# B&R Automation Studio project MotionTestBenchMaster (part 17)

### HMI_PAM_3.typ
```iecst
(*HMI_PAM_3 Database for Filler PLC*)
(*Author = ????*)
(*DB Version : 0.00*)
(*File Version : 3.23*)

TYPE
        HMI_PAM_3_Type:     STRUCT
                            _000 : REAL; (*SEAMER FERRUM - Seamer rinse: Hot water temperature [°C]*)
                            _001 : REAL; (*SEAMER FERRUM - Spare *)
                            _002 : REAL; (*SEAMER FERRUM - Spare *)
                            _003 : REAL; (*SEAMER FERRUM - Spare *)
                            _004 : REAL; (*SEAMER FERRUM - Spare *)
                            _005 : REAL; (*SEAMER FERRUM - Spare *)
                            _006 : REAL; (*SEAMER FERRUM - Spare *)
                            _007 : REAL; (*SEAMER FERRUM - Spare *)
                            _008 : REAL; (*SEAMER FERRUM - Spare *)
                            _009 : REAL; (*SEAMER FERRUM - Spare *)
                            _010 : REAL; (*SEAMER FERRUM - Machine Speed on seamer cleaning [c/h]*)
                            _011 : REAL; (*SEAMER FERRUM - Spare *)
                            _012 : REAL; (*SEAMER FERRUM - Spare *)
                            _013 : REAL; (*SEAMER FERRUM - Spare *)
                            _014 : REAL; (*SEAMER FERRUM - Spare *)
                            _015 : REAL; (*SEAMER FERRUM - Spare *)
                            _016 : REAL; (*SEAMER FERRUM - Spare *)
                            _017 : REAL; (*SEAMER FERRUM - Spare *)
                            _018 : REAL; (*SEAMER FERRUM - Spare *)
                            _019 : REAL; (*SEAMER FERRUM - Spare *)
                            _020 : REAL; (*SEAMER FERRUM - Spare *)
                            _021 : REAL; (*SEAMER FERRUM - Spare *)
                            _022 : REAL; (*SEAMER FERRUM - Spare *)
                            _023 : REAL; (*SEAMER FERRUM - Spare *)
                            _024 : REAL; (*SEAMER FERRUM - Spare *)
                            _025 : REAL; (*SEAMER FERRUM - Spare *)
                            _026 : REAL; (*SEAMER FERRUM - Spare *)
                            _027 : REAL; (*SEAMER FERRUM - Spare *)
                            _028 : REAL; (*SEAMER FERRUM - Spare *)
                            _029 : REAL; (*SEAMER FERRUM - Spare *)
                            _030 : REAL; (*SEAMER FERRUM - Spare *)
                            _031 : REAL; (*SEAMER FERRUM - Spare *)
                            _032 : REAL; (*SEAMER FERRUM - Spare *)
                            _033 : REAL; (*SEAMER FERRUM - Spare *)
                            _034 : REAL; (*SEAMER FERRUM - Spare *)
                            _035 : REAL; (*SEAMER FERRUM - Spare *)
                            _036 : REAL; (*SEAMER FERRUM - Spare *)
                            _037 : REAL; (*SEAMER FERRUM - Spare *)
                            _038 : REAL; (*SEAMER FERRUM - Spare *)
                            _039 : REAL; (*SEAMER FERRUM - Spare *)
                            _040 : REAL; (*SEAMER FERRUM - Spare *)
                            _041 : REAL; (*SEAMER FERRUM - Spare *)
                            _042 : REAL; (*SEAMER FERRUM - Spare *)
                            _043 : REAL; (*SEAMER FERRUM - Spare *)
                            _044 : REAL; (*SEAMER FERRUM - Spare *)
                            _045 : REAL; (*SEAMER FERRUM - Spare *)
                            _046 : REAL; (*SEAMER FERRUM - Spare *)
                            _047 : REAL; (*SEAMER FERRUM - Spare *)
                            _048 : REAL; (*SEAMER FERRUM - Spare *)
                            _049 : REAL; (*SEAMER FERRUM - Spare *)
                            _050 : REAL; (*SEAMER FERRUM - Spare *)
                            _051 : REAL; (*SEAMER FERRUM - Spare *)
                            _052 : REAL; (*SEAMER FERRUM - Spare *)
                            _053 : REAL; (*SEAMER FERRUM - Spare *)
                            _054 : REAL; (*SEAMER FERRUM - Spare *)
                            _055 : REAL; (*SEAMER FERRUM - Spare *)
                            _056 : REAL; (*SEAMER FERRUM - Spare *)
                            _057 : REAL; (*SEAMER FERRUM - Spare *)
                            _058 : REAL; (*SEAMER FERRUM - Spare *)
                            _059 : REAL; (*SEAMER FERRUM - Spare *)
                            _060 : REAL; (*SEAMER FERRUM - Spare *)
                            _061 : REAL; (*SEAMER FERRUM - Spare *)
                            _062 : REAL; (*SEAMER FERRUM - Spare *)
                            _063 : REAL; (*SEAMER FERRUM - Spare *)
                            _064 : REAL; (*SEAMER FERRUM - Spare *)
                            _065 : REAL; (*SEAMER FERRUM - Spare *)
                            _066 : REAL; (*SEAMER FERRUM - Spare *)
                            _067 : REAL; (*SEAMER FERRUM - Spare *)
                            _068 : REAL; (*SEAMER FERRUM - Spare *)
                            _069 : REAL; (*SEAMER FERRUM - Spare *)
                            _070 : REAL; (*SEAMER FERRUM - Spare *)
                            _071 : REAL; (*SEAMER FERRUM - Spare *)
                            _072 : REAL; (*SEAMER FERRUM - Spare *)
                            _073 : REAL; (*SEAMER FERRUM - Spare *)
                            _074 : REAL; (*SEAMER FERRUM - Spare *)
                            _075 : REAL; (*SEAMER FERRUM - Spare *)
                            _076 : REAL; (*SEAMER FERRUM - Spare *)
                            _077 : REAL; (*SEAMER FERRUM - Spare *)
                            _078 : REAL; (*SEAMER FERRUM - Spare *)
                            _079 : REAL; (*SEAMER FERRUM - Spare *)
                            _080 : REAL; (*SEAMER FERRUM - Spare *)
                            _081 : REAL; (*SEAMER FERRUM - Spare *)
                            _082 : REAL; (*SEAMER FERRUM - Spare *)
                            _083 : REAL; (*SEAMER FERRUM - Spare *)
                            _084 : REAL; (*SEAMER FERRUM - Spare *)
                            _085 : REAL; (*SEAMER FERRUM - Spare *)
                            _086 : REAL; (*SEAMER FERRUM - Spare *)
                            _087 : REAL; (*SEAMER FERRUM - Spare *)
                            _088 : REAL; (*SEAMER FERRUM - Spare *)
                            _089 : REAL; (*SEAMER FERRUM - Spare *)
                            _090 : REAL; (*SEAMER FERRUM - Spare *)
                            _091 : REAL; (*SEAMER FERRUM - Spare *)
                            _092 : REAL; (*SEAMER FERRUM - Spare *)
                            _093 : REAL; (*SEAMER FERRUM - Spare *)
                            _094 : REAL; (*SEAMER FERRUM - Spare *)
                            _095 : REAL; (*SEAMER FERRUM - Spare *)
                            _096 : REAL; (*SEAMER FERRUM - Spare *)
                            _097 : REAL; (*SEAMER FERRUM - Spare *)
                            _098 : REAL; (*SEAMER FERRUM - Spare *)
                            _099 : REAL; (*SEAMER FERRUM - Spare *)
                            _100 : REAL; (*SEAMER CFT - Seamer Lubrication *)
                            _101 : REAL; (*SEAMER CFT - Seamer Roll Lubrication *)
                            _102 : REAL; (*SEAMER CFT - Seamer Star Washing Time [s]*)
                            _103 : REAL; (*SEAMER CFT - Seamer Washing Time [s]*)
                            _104 : REAL; (*SEAMER CFT - Low Lubrication Cycle Aft Was *)
                            _105 : REAL; (*SEAMER CFT - Low Lubrication Cycle *)
                            _106 : REAL; (*SEAMER CFT - Lubrication Cycle Aft Was *)
                            _107 : REAL; (*SEAMER CFT - Rol Lubric Cycle *)
                            _108 : REAL; (*SEAMER CFT - N Timer *)
                            _109 : REAL; (*SEAMER CFT - Timer Value *)
                            _110 : REAL; (*SEAMER CFT - Spare *)
                            _111 : REAL; (*SEAMER CFT - Spare *)
                            _112 : REAL; (*SEAMER CFT - Roll_Lubrication_Enable *)
                            _113 : REAL; (*SEAMER CFT - Star Washing Enable *)
                            _114 : REAL; (*SEAMER CFT - Spare *)
                            _115 : REAL; (*SEAMER CFT - Spare *)
                            _116 : REAL; (*SEAMER CFT - Spare *)
                            _117 : REAL; (*SEAMER CFT - Spare *)
                            _118 : REAL; (*SEAMER CFT - Spare *)
                            _119 : REAL; (*SEAMER CFT - Spare *)
                            _120 : REAL; (*SEAMER CFT - Spare *)
                            _121 : REAL; (*SEAMER CFT - Spare *)
                            _122 : REAL; (*SEAMER CFT - Spare *)
                            _123 : REAL; (*SEAMER CFT - Spare *)
                            _124 : REAL; (*SEAMER CFT - Spare *)
                            _125 : REAL; (*SEAMER CFT - Spare *)
                            _126 : REAL; (*SEAMER CFT - Spare *)
                            _127 : REAL; (*SEAMER CFT - Spare *)
                            _128 : REAL; (*SEAMER CFT - Spare *)
                            _129 : REAL; (*SEAMER CFT - Spare *)
                            _130 : REAL; (*SEAMER CFT - Spare *)
                            _131 : REAL; (*SEAMER CFT - Spare *)
                            _132 : REAL; (*SEAMER CFT - Spare *)
                            _133 : REAL; (*SEAMER CFT - Spare *)
                            _134 : REAL; (*SEAMER CFT - Spare *)
                            _135 : REAL; (*SEAMER CFT - Spare *)
                            _136 : REAL; (*SEAMER CFT - Spare *)
                            _137 : REAL; (*SEAMER CFT - Spare *)
                            _138 : REAL; (*SEAMER CFT - Spare *)
                            _139 : REAL; (*SEAMER CFT - Spare *)
                            _140 : REAL; (*SEAMER CFT - Spare *)
                            _141 : REAL; (*SEAMER CFT - Spare *)
                            _142 : REAL; (*SEAMER CFT - Spare *)
                            _143 : REAL; (*SEAMER CFT - Spare *)
                            _144 : REAL; (*SEAMER CFT - Spare *)
                            _145 : REAL; (*SEAMER CFT - Spare *)
                            _146 : REAL; (*SEAMER CFT - Spare *)
                            _147 : REAL; (*SEAMER CFT - Spare *)
                            _148 : REAL; (*SEAMER CFT - Spare *)
                            _149 : REAL; (*SEAMER CFT - Spare *)
                            _150 : REAL; (*SEAMER CFT - Spare *)
                            _151 : REAL; (*SEAMER CFT - Spare *)
                            _152 : REAL; (*SEAMER CFT - Spare *)
                            _153 : REAL; (*SEAMER CFT - Spare *)
                            _154 : REAL; (*SEAMER CFT - Spare *)
                            _155 : REAL; (*SEAMER CFT - Spare *)
                            _156 : REAL; (*SEAMER CFT - Spare *)
                            _157 : REAL; (*SEAMER CFT - Spare *)
                            _158 : REAL; (*SEAMER CFT - Spare *)
                            _159 : REAL; (*SEAMER CFT - Spare *)
                            _160 : REAL; (*SEAMER CFT - Spare *)
                            _161 : REAL; (*SEAMER CFT - Spare *)
                            _162 : REAL; (*SEAMER CFT - Spare *)
                            _163 : REAL; (*SEAMER CFT - Spare *)
                            _164 : REAL; (*SEAMER CFT - Spare *)
                            _165 : REAL; (*SEAMER CFT - Spare *)
                            _166 : REAL; (*SEAMER CFT - Spare *)
                            _167 : REAL; (*SEAMER CFT - Spare *)
                            _168 : REAL; (*SEAMER CFT - Spare *)
                            _169 : REAL; (*SEAMER CFT - Spare *)
                            _170 : REAL; (*SEAMER CFT - Spare *)
                            _171 : REAL; (*SEAMER CFT - Spare *)
                            _172 : REAL; (*SEAMER CFT - Spare *)
                            _173 : REAL; (*SEAMER CFT - Spare *)
                            _174 : REAL; (*SEAMER CFT - Spare *)
                            _175 : REAL; (*SEAMER CFT - Spare *)
                            _176 : REAL; (*SEAMER CFT - Spare *)
                            _177 : REAL; (*SEAMER CFT - Spare *)
                            _178 : REAL; (*SEAMER CFT - Spare *)
                            _179 : REAL; (*SEAMER CFT - Spare *)
                            _180 : REAL; (*SEAMER CFT - Spare *)
                            _181 : REAL; (*SEAMER CFT - Spare *)
                            _182 : REAL; (*SEAMER CFT - Spare *)
                            _183 : REAL; (*SEAMER CFT - Spare *)
                            _184 : REAL; (*SEAMER CFT - Spare *)
                            _185 : REAL; (*SEAMER CFT - Spare *)
                            _186 : REAL; (*SEAMER CFT - Spare *)
                            _187 : REAL; (*SEAMER CFT - Spare *)
                            _188 : REAL; (*SEAMER CFT - Spare *)
                            _189 : REAL; (*SEAMER CFT - Spare *)
                            _190 : REAL; (*SEAMER CFT - Spare *)
                            _191 : REAL; (*SEAMER CFT - Spare *)
                            _192 : REAL; (*SEAMER CFT - Spare *)
                            _193 : REAL; (*SEAMER CFT - Spare *)
                            _194 : REAL; (*SEAMER CFT - Spare *)
                            _195 : REAL; (*SEAMER CFT - Spare *)
                            _196 : REAL; (*SEAMER CFT - Spare *)
                            _197 : REAL; (*SEAMER CFT - Spare *)
                            _198 : REAL; (*SEAMER CFT - Spare *)
                            _199 : REAL; (*SEAMER CFT - Spare *)
                            _200 : REAL; (*SEAMER ANGELUS - Seamer rinse: Hot water temperature [°C]*)
                            _201 : REAL; (*SEAMER ANGELUS - Spare *)
                            _202 : REAL; (*SEAMER ANGELUS - Spare *)
                            _203 : REAL; (*SEAMER ANGELUS - Spare *)
                            _204 : REAL; (*SEAMER ANGELUS - Spare *)
                            _205 : REAL; (*SEAMER ANGELUS - Spare *)
                            _206 : REAL; (*SEAMER ANGELUS - Spare *)
                            _207 : REAL; (*SEAMER ANGELUS - Spare *)
                            _208 : REAL; (*SEAMER ANGELUS - Spare *)
                            _209 : REAL; (*SEAMER ANGELUS - Spare *)
                            _210 : REAL; (*SEAMER ANGELUS - Machine Speed on seamer cleaning [c/h]*)
                            _211 : REAL; (*SEAMER ANGELUS - Spare *)
                            _212 : REAL; (*SEAMER ANGELUS - Spare *)
                            _213 : REAL; (*SEAMER ANGELUS - Spare *)
                            _214 : REAL; (*SEAMER ANGELUS - Spare *)
                            _215 : REAL; (*SEAMER ANGELUS - Spare *)
                            _216 : REAL; (*SEAMER ANGELUS - Spare *)
                            _217 : REAL; (*SEAMER ANGELUS - Spare *)
                            _218 : REAL; (*SEAMER ANGELUS - Spare *)
                            _219 : REAL; (*SEAMER ANGELUS - Spare *)
                            _220 : REAL; (*SEAMER ANGELUS - Spare *)
                            _221 : REAL; (*SEAMER ANGELUS - Spare *)
                            _222 : REAL; (*SEAMER ANGELUS - Spare *)
                            _223 : REAL; (*SEAMER ANGELUS - Spare *)
                            _224 : REAL; (*SEAMER ANGELUS - Spare *)
                            _225 : REAL; (*SEAMER ANGELUS - Spare *)
                            _226 : REAL; (*SEAMER ANGELUS - Spare *)
                            _227 : REAL; (*SEAMER ANGELUS - Spare *)
                            _228 : REAL; (*SEAMER ANGELUS - Spare *)
                            _229 : REAL; (*SEAMER ANGELUS - Spare *)
                            _230 : REAL; (*SEAMER ANGELUS - Spare *)
                            _231 : REAL; (*SEAMER ANGELUS - Spare *)
                            _232 : REAL; (*SEAMER ANGELUS - Spare *)
                            _233 : REAL; (*SEAMER ANGELUS - Spare *)
                            _234 : REAL; (*SEAMER ANGELUS - Spare *)
                            _235 : REAL; (*SEAMER ANGELUS - Spare *)
                            _236 : REAL; (*SEAMER ANGELUS - Spare *)
                            _237 : REAL; (*SEAMER ANGELUS - Spare *)
                            _238 : REAL; (*SEAMER ANGELUS - Spare *)
                            _239 : REAL; (*SEAMER ANGELUS - Spare *)
                            _240 : REAL; (*SEAMER ANGELUS - Spare *)
                            _241 : REAL; (*SEAMER ANGELUS - Spare *)
                            _242 : REAL; (*SEAMER ANGELUS - Spare *)
                            _243 : REAL; (*SEAMER ANGELUS - Spare *)
                            _244 : REAL; (*SEAMER ANGELUS - Spare *)
                            _245 : REAL; (*SEAMER ANGELUS - Spare *)
                            _246 : REAL; (*SEAMER ANGELUS - Spare *)
                            _247 : REAL; (*SEAMER ANGELUS - Spare *)
                            _248 : REAL; (*SEAMER ANGELUS - Spare *)
                            _249 : REAL; (*SEAMER ANGELUS - Spare *)
                            _250 : REAL; (*SEAMER ANGELUS - Spare *)
                            _251 : REAL; (*SEAMER ANGELUS - Spare *)
                            _252 : REAL; (*SEAMER ANGELUS - Spare *)
                            _253 : REAL; (*SEAMER ANGELUS - Spare *)
                            _254 : REAL; (*SEAMER ANGELUS - Spare *)
                            _255 : REAL; (*SEAMER ANGELUS - Spare *)
                            _256 : REAL; (*SEAMER ANGELUS - Spare *)
                            _257 : REAL; (*SEAMER ANGELUS - Spare *)
                            _258 : REAL; (*SEAMER ANGELUS - Spare *)
                            _259 : REAL; (*SEAMER ANGELUS - Spare *)
                            _260 : REAL; (*SEAMER ANGELUS - Spare *)
                            _261 : REAL; (*SEAMER ANGELUS - Spare *)
                            _262 : REAL; (*SEAMER ANGELUS - Spare *)
                            _263 : REAL; (*SEAMER ANGELUS - Spare *)
                            _264 : REAL; (*SEAMER ANGELUS - Spare *)
                            _265 : REAL; (*SEAMER ANGELUS - Spare *)
                            _266 : REAL; (*SEAMER ANGELUS - Spare *)
                            _267 : REAL; (*SEAMER ANGELUS - Spare *)
                            _268 : REAL; (*SEAMER ANGELUS - Spare *)
                            _269 : REAL; (*SEAMER ANGELUS - Spare *)
                            _270 : REAL; (*SEAMER ANGELUS - Spare *)
                            _271 : REAL; (*SEAMER ANGELUS - Spare *)
                            _272 : REAL; (*SEAMER ANGELUS - Spare *)
                            _273 : REAL; (*SEAMER ANGELUS - Spare *)
                            _274 : REAL; (*SEAMER ANGELUS - Spare *)
                            _275 : REAL; (*SEAMER ANGELUS - Spare *)
                            _276 : REAL; (*SEAMER ANGELUS - Spare *)
                            _277 : REAL; (*SEAMER ANGELUS - Spare *)
                            _278 : REAL; (*SEAMER ANGELUS - Spare *)
                            _279 : REAL; (*SEAMER ANGELUS - Spare *)
                            _280 : REAL; (*SEAMER ANGELUS - Spare *)
                            _281 : REAL; (*SEAMER ANGELUS - Spare *)
                            _282 : REAL; (*SEAMER ANGELUS - Spare *)
                            _283 : REAL; (*SEAMER ANGELUS - Spare *)
                            _284 : REAL; (*SEAMER ANGELUS - Spare *)
                            _285 : REAL; (*SEAMER ANGELUS - Spare *)
                            _286 : REAL; (*SEAMER ANGELUS - Spare *)
                            _287 : REAL; (*SEAMER ANGELUS - Spare *)
                            _288 : REAL; (*SEAMER ANGELUS - Spare *)
                            _289 : REAL; (*SEAMER ANGELUS - Spare *)
                            _290 : REAL; (*SEAMER ANGELUS - Spare *)
                            _291 : REAL; (*SEAMER ANGELUS - Spare *)
                            _292 : REAL; (*SEAMER ANGELUS - Spare *)
                            _293 : REAL; (*SEAMER ANGELUS - Spare *)
                            _294 : REAL; (*SEAMER ANGELUS - Spare *)
                            _295 : REAL; (*SEAMER ANGELUS - Spare *)
                            _296 : REAL; (*SEAMER ANGELUS - Spare *)
                            _297 : REAL; (*SEAMER ANGELUS - Spare *)
                            _298 : REAL; (*SEAMER ANGELUS - Spare *)
                            _299 : REAL; (*SEAMER ANGELUS - Spare *)
                            _300 : REAL; (*RINSER - Spare *)
                            _301 : REAL; (*RINSER - Spare *)
                            _302 : REAL; (*RINSER - Spare *)
                            _303 : REAL; (*RINSER - Spare *)
                            _304 : REAL; (*RINSER - Spare *)
                            _305 : REAL; (*RINSER - Spare *)
                            _306 : REAL; (*RINSER - Spare *)
                            _307 : REAL; (*RINSER - Spare *)
                            _308 : REAL; (*RINSER - Spare *)
                            _309 : REAL; (*RINSER - Spare *)
                            _310 : REAL; (*RINSER - Spare *)
                            _311 : REAL; (*RINSER - Spare *)
                            _312 : REAL; (*RINSER - Spare *)
                            _313 : REAL; (*RINSER - Spare *)
                            _314 : REAL; (*RINSER - Spare *)
                            _315 : REAL; (*RINSER - Spare *)
                            _316 : REAL; (*RINSER - Spare *)
                            _317 : REAL; (*RINSER - Spare *)
                            _318 : REAL; (*RINSER - Spare *)
                            _319 : REAL; (*RINSER - Spare *)
                            _320 : REAL; (*RINSER - Spare *)
                            _321 : REAL; (*RINSER - Spare *)
                            _322 : REAL; (*RINSER - Spare *)
                            _323 : REAL; (*RINSER - Spare *)
                            _324 : REAL; (*RINSER - Spare *)
                            _325 : REAL; (*RINSER - Spare *)
                            _326 : REAL; (*RINSER - Spare *)
                            _327 : REAL; (*RINSER - Spare *)
                            _328 : REAL; (*RINSER - Spare *)
                            _329 : REAL; (*RINSER - Spare *)
                            _330 : REAL; (*RINSER - Spare *)
                            _331 : REAL; (*RINSER - Spare *)
                            _332 : REAL; (*RINSER - Spare *)
                            _333 : REAL; (*RINSER - Spare *)
                            _334 : REAL; (*RINSER - Spare *)
                            _335 : REAL; (*RINSER - Spare *)
                            _336 : REAL; (*RINSER - Spare *)
                            _337 : REAL; (*RINSER - Spare *)
                            _338 : REAL; (*RINSER - Spare *)
                            _339 : REAL; (*RINSER - Spare *)
                            _340 : REAL; (*RINSER - Spare *)
                            _341 : REAL; (*RINSER - Spare *)
                            _342 : REAL; (*RINSER - Spare *)
                            _343 : REAL; (*RINSER - Spare *)
                            _344 : REAL; (*RINSER - Spare *)
                            _345 : REAL; (*RINSER - Spare *)
                            _346 : REAL; (*RINSER - Spare *)
                            _347 : REAL; (*RINSER - Spare *)
                            _348 : REAL; (*RINSER - Spare *)
                            _349 : REAL; (*RINSER - Spare *)
                            _350 : REAL; (*RINSER - Spare *)
                            _351 : REAL; (*RINSER - Spare *)
                            _352 : REAL; (*RINSER - Spare *)
                            _353 : REAL; (*RINSER - Spare *)
                            _354 : REAL; (*RINSER - Spare *)
                            _355 : REAL; (*RINSER - Spare *)
                            _356 : REAL; (*RINSER - Spare *)
                            _357 : REAL; (*RINSER - Spare *)
                            _358 : REAL; (*RINSER - Spare *)
                            _359 : REAL; (*RINSER - Spare *)
                            _360 : REAL; (*RINSER - Spare *)
                            _361 : REAL; (*RINSER - Spare *)
                            _362 : REAL; (*RINSER - Spare *)
                            _363 : REAL; (*RINSER - Spare *)
                            _364 : REAL; (*RINSER - Spare *)
                            _365 : REAL; (*RINSER - Spare *)
                            _366 : REAL; (*RINSER - Spare *)
                            _367 : REAL; (*RINSER - Spare *)
                            _368 : REAL; (*RINSER - Spare *)
                            _369 : REAL; (*RINSER - Spare *)
                            _370 : REAL; (*RINSER - Spare *)
                            _371 : REAL; (*RINSER - Spare *)
                            _372 : REAL; (*RINSER - Spare *)
                            _373 : REAL; (*RINSER - Spare *)
                            _374 : REAL; (*RINSER - Spare *)
                            _375 : REAL; (*RINSER - Spare *)
                            _376 : REAL; (*RINSER - Spare *)
                            _377 : REAL; (*RINSER - Spare *)
                            _378 : REAL; (*RINSER - Spare *)
                            _379 : REAL; (*RINSER - Spare *)
                            _380 : REAL; (*RINSER - Spare *)
                            _381 : REAL; (*RINSER - Spare *)
                            _382 : REAL; (*RINSER - Spare *)
                            _383 : REAL; (*RINSER - Spare *)
                            _384 : REAL; (*RINSER - Spare *)
                            _385 : REAL; (*RINSER - Spare *)
                            _386 : REAL; (*RINSER - Spare *)
                            _387 : REAL; (*RINSER - Spare *)
                            _388 : REAL; (*RINSER - Spare *)
                            _389 : REAL; (*RINSER - Spare *)
                            _390 : REAL; (*RINSER - Spare *)
                            _391 : REAL; (*RINSER - Spare *)
                            _392 : REAL; (*RINSER - Spare *)
                            _393 : REAL; (*RINSER - Spare *)
                            _394 : REAL; (*RINSER - Spare *)
                            _395 : REAL; (*RINSER - Spare *)
                            _396 : REAL; (*RINSER - Spare *)
                            _397 : REAL; (*RINSER - Spare *)
                            _398 : REAL; (*RINSER - Spare *)
                            _399 : REAL; (*RINSER - Spare *)
                            _400 : REAL; (*CROWNER - Max Number of missing Caps in the Channel *)
                            _401 : REAL; (*CROWNER - Max Number of missing Caps in the Starweel *)
                            _402 : REAL; (*CROWNER - Spare *)
                            _403 : REAL; (*CROWNER - Spare *)
                            _404 : REAL; (*CROWNER - Spare *)
                            _405 : REAL; (*CROWNER - Spare *)
                            _406 : REAL; (*CROWNER - Spare *)
                            _407 : REAL; (*CROWNER - Spare *)
                            _408 : REAL; (*CROWNER - Spare *)
                            _409 : REAL; (*CROWNER - Spare *)
                            _410 : REAL; (*CROWNER - Lifting Crowner Sensor Position Offset *)
                            _411 : REAL; (*CROWNER - Spare *)
                            _412 : REAL; (*CROWNER - Spare *)
                            _413 : REAL; (*CROWNER - Spare *)
                            _414 : REAL; (*CROWNER - Spare *)
                            _415 : REAL; (*CROWNER - Spare *)
                            _416 : REAL; (*CROWNER - Spare *)
                            _417 : REAL; (*CROWNER - Spare *)
                            _418 : REAL; (*CROWNER - Spare *)
                            _419 : REAL; (*CROWNER - Spare *)
                            _420 : REAL; (*CROWNER - Spare *)
                            _421 : REAL; (*CROWNER - Spare *)
                            _422 : REAL; (*CROWNER - Spare *)
                            _423 : REAL; (*CROWNER - Spare *)
                            _424 : REAL; (*CROWNER - Spare *)
                            _425 : REAL; (*CROWNER - Spare *)
                            _426 : REAL; (*CROWNER - Spare *)
                            _427 : REAL; (*CROWNER - Spare *)
                            _428 : REAL; (*CROWNER - Spare *)
                            _429 : REAL; (*CROWNER - Spare *)
                            _430 : REAL; (*CROWNER - Spare *)
                            _431 : REAL; (*CROWNER - Spare *)
                            _432 : REAL; (*CROWNER - Spare *)
                            _433 : REAL; (*CROWNER - Spare *)
                            _434 : REAL; (*CROWNER - Spare *)
                            _435 : REAL; (*CROWNER - Spare *)
                            _436 : REAL; (*CROWNER - Spare *)
                            _437 : REAL; (*CROWNER - Spare *)
                            _438 : REAL; (*CROWNER - Spare *)
                            _439 : REAL; (*CROWNER - Spare *)
                            _440 : REAL; (*CROWNER - Spare *)
                            _441 : REAL; (*CROWNER - Spare *)
                            _442 : REAL; (*CROWNER - Spare *)
                            _443 : REAL; (*CROWNER - Spare *)
                            _444 : REAL; (*CROWNER - Spare *)
                            _445 : REAL; (*CROWNER - Spare *)
                            _446 : REAL; (*CROWNER - Spare *)
                            _447 : REAL; (*CROWNER - Spare *)
                            _448 : REAL; (*CROWNER - Spare *)
                            _449 : REAL; (*CROWNER - Spare *)
                            _450 : REAL; (*CROWNER - Spare *)
                            _451 : REAL; (*CROWNER - Spare *)
                            _452 : REAL; (*CROWNER - Spare *)
                            _453 : REAL; (*CROWNER - Spare *)
                            _454 : REAL; (*CROWNER - Spare *)
                            _455 : REAL; (*CROWNER - Spare *)
                            _456 : REAL; (*CROWNER - Spare *)
                            _457 : REAL; (*CROWNER - Spare *)
                            _458 : REAL; (*CROWNER - Spare *)
                            _459 : REAL; (*CROWNER - Spare *)
                            _460 : REAL; (*CROWNER - Spare *)
                            _461 : REAL; (*CROWNER - Spare *)
                            _462 : REAL; (*CROWNER - Spare *)
                            _463 : REAL; (*CROWNER - Spare *)
                            _464 : REAL; (*CROWNER - Spare *)
                            _465 : REAL; (*CROWNER - Spare *)
                            _466 : REAL; (*CROWNER - Spare *)
                            _467 : REAL; (*CROWNER - Spare *)
                            _468 : REAL; (*CROWNER - Spare *)
                            _469 : REAL; (*CROWNER - Spare *)
                            _470 : REAL; (*CROWNER - Spare *)
                            _471 : REAL; (*CROWNER - Spare *)
                            _472 : REAL; (*CROWNER - Spare *)
                            _473 : REAL; (*CROWNER - Spare *)
                            _474 : REAL; (*CROWNER - Spare *)
                            _475 : REAL; (*CROWNER - Spare *)
                            _476 : REAL; (*CROWNER - Spare *)
                            _477 : REAL; (*CROWNER - Spare *)
                            _478 : REAL; (*CROWNER - Spare *)
                            _479 : REAL; (*CROWNER - Spare *)
                            _480 : REAL; (*CROWNER - Spare *)
                            _481 : REAL; (*CROWNER - Spare *)
                            _482 : REAL; (*CROWNER - Spare *)
                            _483 : REAL; (*CROWNER - Spare *)
                            _484 : REAL; (*CROWNER - Spare *)
                            _485 : REAL; (*CROWNER - Spare *)
                            _486 : REAL; (*CROWNER - Spare *)
                            _487 : REAL; (*CROWNER - Spare *)
                            _488 : REAL; (*CROWNER - Spare *)
                            _489 : REAL; (*CROWNER - Spare *)
                            _490 : REAL; (*CROWNER - Spare *)
                            _491 : REAL; (*CROWNER - Spare *)
                            _492 : REAL; (*CROWNER - Spare *)
                            _493 : REAL; (*CROWNER - Spare *)
                            _494 : REAL; (*CROWNER - Spare *)
                            _495 : REAL; (*CROWNER - Spare *)
                            _496 : REAL; (*CROWNER - Spare *)
                            _497 : REAL; (*CROWNER - Spare *)
                            _498 : REAL; (*CROWNER - Spare *)
                            _499 : REAL; (*CROWNER - Spare *)
                            _500 : REAL; (*CAPPER - Max Number of missing Caps in the Channel *)
                            _501 : REAL; (*CAPPER - Max Number of missing Caps in the Starweel - Consecutive Error *)
                            _502 : REAL; (*CAPPER - Max Number of Head Consecutive Error *)
                            _503 : REAL; (*CAPPER - Max Number of Total Consecutive Error *)
                            _504 : REAL; (*CAPPER - Number of caps for absolute control *)
                            _505 : REAL; (*CAPPER - Max Number of missing Caps in the Starweel - Bottle Stop *)
                            _506 : REAL; (*CAPPER - Max Number of missing Caps in the Bottle - Consecutive Error *)
                            _507 : REAL; (*CAPPER - Number of Uncapped Bottles for absolute control *)
                            _508 : REAL; (*CAPPER - Max Number Uncapped Bottle *)
                            _509 : REAL; (*CAPPER - Spare *)
                            _510 : REAL; (*CAPPER - HRM CW Head Rotation *)
                            _511 : REAL; (*CAPPER - HRM GearIn *)
                            _512 : REAL; (*CAPPER - HRM GearOut *)
                            _513 : REAL; (*CAPPER - HRM Missing Caps number in the starwheel before alarm *)
                            _514 : REAL; (*CAPPER - Spare *)
                            _515 : REAL; (*CAPPER - Spare *)
                            _516 : REAL; (*CAPPER - Spare *)
                            _517 : REAL; (*CAPPER - Spare *)
                            _518 : REAL; (*CAPPER - Spare *)
                            _519 : REAL; (*CAPPER - Spare *)
                            _520 : REAL; (*CAPPER - Sterilizer Wet: Caps inside the channel *)
                            _521 : REAL; (*CAPPER - Sterilizer Wet: Number of caps before slidind fault *)
                            _522 : REAL; (*CAPPER - Spare *)
                            _523 : REAL; (*CAPPER - Spare *)
                            _524 : REAL; (*CAPPER - Spare *)
                            _525 : INT; (*CAPPER - Greasing cycle number [unit]*)
                            _526 : INT; (*CAPPER - Greasing request hours [h]*)
                            _527 : INT; (*CAPPER - Greasing cycle timeout [s]*)
                            _528 : REAL; (*CAPPER - Greasing sensor position offset [mm]*)
                            _529 : REAL; (*CAPPER - Greasing flow alarm timeout [s]*)
                            _530 : REAL; (*CAPPER - Greasing cycle number (2nd Pump) [unit]*)
                            _531 : REAL; (*CAPPER - Greasing request hours (2nd Pump) [h]*)
                            _532 : REAL; (*CAPPER - Greasing cycle timeout (2nd Pump) [s]*)
                            _533 : REAL; (*CAPPER - Spare *)
                            _534 : REAL; (*CAPPER - Greasing flow alarm timeout (2nd Pump) [s]*)
                            _535 : REAL; (*CAPPER - Spare *)
                            _536 : REAL; (*CAPPER - Spare *)
                            _537 : REAL; (*CAPPER - Spare *)
                            _538 : REAL; (*CAPPER - Spare *)
                            _539 : REAL; (*CAPPER - Spare *)
                            _540 : REAL; (*CAPPER - Lifting Capper Sensor Position Offset [mm]*)
                            _541 : REAL; (*CAPPER - Spare *)
                            _542 : REAL; (*CAPPER - Spare *)
                            _543 : REAL; (*CAPPER - Spare *)
                            _544 : REAL; (*CAPPER - Spare *)
                            _545 : REAL; (*CAPPER - Spare *)
                            _546 : REAL; (*CAPPER - Spare *)
                            _547 : REAL; (*CAPPER - Spare *)
                            _548 : REAL; (*CAPPER - Spare *)
                            _549 : REAL; (*CAPPER - Spare *)
                            _550 : REAL; (*CAPPER - Hopper 1 Drive - OUT Min [%]*)
                            _551 : REAL; (*CAPPER - Hopper 1 Drive - OUT Max [%]*)
                            _552 : REAL; (*CAPPER - Hopper 1 Drive - Spare *)
                            _553 : REAL; (*CAPPER - Hopper 1 Drive - Spare *)
                            _554 : REAL; (*CAPPER - Hopper 2 Drive - OUT Min [%]*)
                            _555 : REAL; (*CAPPER - Hopper 2 Drive - OUT Max [%]*)
                            _556 : REAL; (*CAPPER - Hopper 2 Drive - Spare *)
                            _557 : REAL; (*CAPPER - Hopper 2 Drive - Spare *)
                            _558 : REAL; (*CAPPER - Hopper 3 Drive - OUT Min [%]*)
                            _559 : REAL; (*CAPPER - Hopper 3 Drive - OUT Max [%]*)
                            _560 : REAL; (*CAPPER - Hopper 3 Drive - Spare *)
                            _561 : REAL; (*CAPPER - Hopper 3 Drive - Spare *)
                            _562 : REAL; (*CAPPER - Hopper 4 Drive - OUT Min [%]*)
                            _563 : REAL; (*CAPPER - Hopper 4 Drive - OUT Max [%]*)
                            _564 : REAL; (*CAPPER - Hopper 4 Drive - Spare *)
                            _565 : REAL; (*CAPPER - Hopper 4 Drive - Spare *)
                            _566 : REAL; (*CAPPER - Head Rotation Drive - OUT Min [%]*)
                            _567 : REAL; (*CAPPER - Head Rotation Drive - OUT Max [%]*)
                            _568 : REAL; (*CAPPER - Head Rotation Drive - Spare *)
                            _569 : REAL; (*CAPPER - Head Rotation Drive - Spare *)
                            _570 : REAL; (*CAPPER - Buffer Drive - OUT Min [%]*)
                            _571 : REAL; (*CAPPER - Buffer Drive - OUT Max [%]*)
                            _572 : REAL; (*CAPPER - Buffer Drive - OUT Min [%]*)
                            _573 : REAL; (*CAPPER - Buffer Drive - OUT Max [%]*)
                            _574 : REAL; (*CAPPER - Buffer Adjustment - OUT Min [%]*)
                            _575 : REAL; (*CAPPER - Buffer Adjustment - OUT Max [%]*)
                            _576 : REAL; (*CAPPER - Spare *)
                            _577 : REAL; (*CAPPER - Spare *)
                            _578 : REAL; (*CAPPER - Spare *)
                            _579 : REAL; (*CAPPER - Spare *)
                            _580 : REAL; (*CAPPER - Spare *)
                            _581 : REAL; (*CAPPER - Spare *)
                            _582 : REAL; (*CAPPER - Spare *)
                            _583 : REAL; (*CAPPER - Spare *)
                            _584 : REAL; (*CAPPER - Spare *)
                            _585 : REAL; (*CAPPER - Spare *)
                            _586 : REAL; (*CAPPER - Spare *)
                            _587 : REAL; (*CAPPER - Spare *)
                            _588 : REAL; (*CAPPER - Spare *)
                            _589 : REAL; (*CAPPER - Spare *)
                            _590 : REAL; (*CAPPER - Spare *)
                            _591 : REAL; (*CAPPER - Spare *)
                            _592 : REAL; (*CAPPER - Spare *)
                            _593 : REAL; (*CAPPER - Spare *)
                            _594 : REAL; (*CAPPER - Spare *)
                            _595 : REAL; (*CAPPER - Spare *)
                            _596 : REAL; (*CAPPER - Spare *)
                            _597 : REAL; (*CAPPER - Spare *)
                            _598 : REAL; (*CAPPER - Spare *)
                            _599 : REAL; (*CAPPER - Spare *)
                            _600 : REAL; (*PulpDoser - Production: Sacs SP [°C]*)
                            _601 : REAL; (*PulpDoser - Production: ICS Tank StartUp Level [%]*)
                            _602 : REAL; (*PulpDoser - Production: Tank StartUp Level [%]*)
                            _603 : REAL; (*PulpDoser - Production: Min Tank Temperature [°C]*)
                            _604 : REAL; (*PulpDoser - Production: Max Tank Temperature [°C]*)
                            _605 : REAL; (*PulpDoser - Production: StartUp Steril Time [s]*)
                            _606 : REAL; (*PulpDoser - Production: Tank Min Lev [%]*)
                            _607 : REAL; (*PulpDoser - Production: Tank Max Lev [%]*)
                            _608 : REAL; (*PulpDoser - Production: Tank SP [%]*)
                            _609 : REAL; (*PulpDoser - Production: Tank Lev OK [%]*)
                            _610 : REAL; (*PulpDoser - Production: Tank Level SP Deviation [%] dev*)
                            _611 : REAL; (*PulpDoser - Heating With Water: PPJ203 - Opening Flip Time  [s]*)
                            _612 : REAL; (*PulpDoser - Heating With Water: PPJ203 - Closing Flip Time  [s]*)
                            _613 : REAL; (*PulpDoser - Heating With Water: AVJ217 - Opening Flip Time  [s]*)
                            _614 : REAL; (*PulpDoser - Heating With Water: AVJ217 - Closing Flip Time [s]*)
                            _615 : REAL; (*PulpDoser - Heating With Water: PPJ202 - Frequency [Hz]*)
                            _616 : REAL; (*PulpDoser - Heating With Water:Time of Circulation at Temperature Reached [s]*)
                            _617 : REAL; (*PulpDoser - Production: Spare *)
                            _618 : REAL; (*PulpDoser - Production: Spare *)
                            _619 : REAL; (*PulpDoser - Production: Spare *)
                            _620 : REAL; (*PulpDoser - Cleaning: Max Tank temperature [°C] dev*)
                            _621 : REAL; (*PulpDoser - Cleaning: Min Tank temperature [°C] dev*)
                            _622 : REAL; (*PulpDoser - Cleaning: Piston Time [s]*)
                            _623 : REAL; (*PulpDoser - Cleaning: Nozzle Time [s]*)
                            _624 : REAL; (*PulpDoser - Cleaning: Drain Time [s]*)
                            _625 : REAL; (*PulpDoser - Cleaning: Conducibility Min [ms]*)
                            _626 : REAL; (*PulpDoser - Cleaning: Tank Level [%]*)
                            _627 : REAL; (*PulpDoser - Cleaning: PPL201 SP [l/min]*)
                            _628 : REAL; (*PulpDoser - Cleaning: PPL201 Min Limit [l/min]*)
                            _629 : REAL; (*PulpDoser - Cleaning: Volume caustic Phase [ml]*)
                            _630 : REAL; (*PulpDoser - Cleaning: PPJ202 Frequency [Hz]*)
                            _631 : REAL; (*PulpDoser - Cleaning: Pulp Doser CIP Speed  [c/h]*)
                            _632 : REAL; (*PulpDoser - Cleaning: Pulp Doser COP Speed  [c/h]*)
                            _633 : REAL; (*PulpDoser - Cleaning: SP Temperature [°C]*)
                            _634 : REAL; (*PulpDoser - Cleaning: PPJ203 - Opening Flip Time  [s]*)
                            _635 : REAL; (*PulpDoser - Cleaning: PPJ203 - Closing Flip Time  [s]*)
                            _636 : REAL; (*PulpDoser - Cleaning: AVJ217 - Opening Flip Time   [s]*)
                            _637 : REAL; (*PulpDoser - Cleaning: AVJ217 - Closing Flip Time  [s]*)
                            _638 : REAL; (*PulpDoser - Cleaning: Spare *)
                            _639 : REAL; (*PulpDoser - Cleaning: Spare *)
                            _640 : REAL; (*PulpDoser - Rinse: Pipe Time [s]*)
                            _641 : REAL; (*PulpDoser - Rinse: Piston Time [s]*)
                            _642 : REAL; (*PulpDoser - Rinse: Piston Wash Cycle  *)
                            _643 : REAL; (*PulpDoser - Rinse: Piston Wash Laps *)
                            _644 : REAL; (*PulpDoser - Rinse: Tank Level [%]*)
                            _645 : REAL; (*PulpDoser - Drain Time [s]*)
                            _646 : REAL; (*PulpDoser - Spare *)
                            _647 : REAL; (*PulpDoser - Spare *)
                            _648 : REAL; (*PulpDoser - Spare *)
                            _649 : REAL; (*PulpDoser - Spare *)
                            _650 : REAL; (*PulpDoser - Spare *)
                            _651 : REAL; (*PulpDoser - Spare *)
                            _652 : REAL; (*PulpDoser - Spare *)
                            _653 : REAL; (*PulpDoser - Spare *)
                            _654 : REAL; (*PulpDoser - Spare *)
                            _655 : REAL; (*PulpDoser - Spare *)
                            _656 : REAL; (*PulpDoser - Spare *)
                            _657 : REAL; (*PulpDoser - Spare *)
                            _658 : REAL; (*PulpDoser - Spare *)
                            _659 : REAL; (*PulpDoser - Spare *)
                            _660 : REAL; (*PulpDoser - Spare *)
                            _661 : REAL; (*PulpDoser - Spare *)
                            _662 : REAL; (*PulpDoser - Spare *)
                            _663 : REAL; (*PulpDoser - Spare *)
                            _664 : REAL; (*PulpDoser - Spare *)
                            _665 : REAL; (*PulpDoser - Spare *)
                            _666 : REAL; (*PulpDoser - Spare *)
                            _667 : REAL; (*PulpDoser - Spare *)
                            _668 : REAL; (*PulpDoser - Spare *)
                            _669 : REAL; (*PulpDoser - Spare *)
                            _670 : REAL; (*PulpDoser - Spare *)
                            _671 : REAL; (*PulpDoser - Spare *)
                            _672 : REAL; (*PulpDoser - Spare *)
                            _673 : REAL; (*PulpDoser - Spare *)
                            _674 : REAL; (*PulpDoser - Spare *)
                            _675 : REAL; (*PulpDoser - Spare *)
                            _676 : REAL; (*PulpDoser - Spare *)
                            _677 : REAL; (*PulpDoser - Spare *)
                            _678 : REAL; (*PulpDoser - Spare *)
                            _679 : REAL; (*PulpDoser - Spare *)
                            _680 : REAL; (*PulpDoser - Spare *)
                            _681 : REAL; (*PulpDoser - Spare *)
                            _682 : REAL; (*PulpDoser - Spare *)
                            _683 : REAL; (*PulpDoser - Spare *)
                            _684 : REAL; (*PulpDoser - Spare *)
                            _685 : REAL; (*PulpDoser - Spare *)
                            _686 : REAL; (*PulpDoser - Spare *)
                            _687 : REAL; (*PulpDoser - Spare *)
                            _688 : REAL; (*PulpDoser - Spare *)
                            _689 : REAL; (*PulpDoser - Spare *)
                            _690 : REAL; (*PulpDoser - Spare *)
                            _691 : REAL; (*PulpDoser - Spare *)
                            _692 : REAL; (*PulpDoser - Spare *)
                            _693 : REAL; (*PulpDoser - Spare *)
                            _694 : REAL; (*PulpDoser - Spare *)
                            _695 : REAL; (*PulpDoser - Spare *)
                            _696 : REAL; (*PulpDoser - Spare *)
                            _697 : REAL; (*PulpDoser - Spare *)
                            _698 : REAL; (*PulpDoser - Spare *)
                            _699 : REAL; (*PulpDoser - Spare *)
                            _700 : REAL; (*SPARE - Spare *)
                            _701 : REAL; (*SPARE - Spare *)
                            _702 : REAL; (*SPARE - Spare *)
                            _703 : REAL; (*SPARE - Spare *)
                            _704 : REAL; (*SPARE - Spare *)
                            _705 : REAL; (*SPARE - Spare *)
                            _706 : REAL; (*SPARE - Spare *)
                            _707 : REAL; (*SPARE - Spare *)
                            _708 : REAL; (*SPARE - Spare *)
                            _709 : REAL; (*SPARE - Spare *)
                            _710 : REAL; (*SPARE - Spare *)
                            _711 : REAL; (*SPARE - Spare *)
                            _712 : REAL; (*SPARE - Spare *)
                            _713 : REAL; (*SPARE - Spare *)
                            _714 : REAL; (*SPARE - Spare *)
                            _715 : REAL; (*SPARE - Spare *)
                            _716 : REAL; (*SPARE - Spare *)
                            _717 : REAL; (*SPARE - Spare *)
                            _718 : REAL; (*SPARE - Spare *)
                            _719 : REAL; (*SPARE - Spare *)
                            _720 : REAL; (*SPARE - Spare *)
                            _721 : REAL; (*SPARE - Spare *)
                            _722 : REAL; (*SPARE - Spare *)
                            _723 : REAL; (*SPARE - Spare *)
                            _724 : REAL; (*SPARE - Spare *)
                            _725 : REAL; (*SPARE - Spare *)
                            _726 : REAL; (*SPARE - Spare *)
                            _727 : REAL; (*SPARE - Spare *)
                            _728 : REAL; (*SPARE - Spare *)
                            _729 : REAL; (*SPARE - Spare *)
                            _730 : REAL; (*SPARE - Spare *)
                            _731 : REAL; (*SPARE - Spare *)
                            _732 : REAL; (*SPARE - Spare *)
                            _733 : REAL; (*SPARE - Spare *)
                            _734 : REAL; (*SPARE - Spare *)
                            _735 : REAL; (*SPARE - Spare *)
                            _736 : REAL; (*SPARE - Spare *)
                            _737 : REAL; (*SPARE - Spare *)
                            _738 : REAL; (*SPARE - Spare *)
                            _739 : REAL; (*SPARE - Spare *)
                            _740 : REAL; (*SPARE - Spare *)
                            _741 : REAL; (*SPARE - Spare *)
                            _742 : REAL; (*SPARE - Spare *)
                            _743 : REAL; (*SPARE - Spare *)
                            _744 : REAL; (*SPARE - Spare *)
                            _745 : REAL; (*SPARE - Spare *)
                            _746 : REAL; (*SPARE - Spare *)
                            _747 : REAL; (*SPARE - Spare *)
                            _748 : REAL; (*SPARE - Spare *)
                            _749 : REAL; (*SPARE - Spare *)
                            _750 : REAL; (*SPARE - Spare *)
                            _751 : REAL; (*SPARE - Spare *)
                            _752 : REAL; (*SPARE - Spare *)
                            _753 : REAL; (*SPARE - Spare *)
                            _754 : REAL; (*SPARE - Spare *)
                            _755 : REAL; (*SPARE - Spare *)
                            _756 : REAL; (*SPARE - Spare *)
                            _757 : REAL; (*SPARE - Spare *)
                            _758 : REAL; (*SPARE - Spare *)
                            _759 : REAL; (*SPARE - Spare *)
                            _760 : REAL; (*SPARE - Spare *)
                            _761 : REAL; (*SPARE - Spare *)
                            _762 : REAL; (*SPARE - Spare *)
                            _763 : REAL; (*SPARE - Spare *)
                            _764 : REAL; (*SPARE - Spare *)
                            _765 : REAL; (*SPARE - Spare *)
                            _766 : REAL; (*SPARE - Spare *)
                            _767 : REAL; (*SPARE - Spare *)
                            _768 : REAL; (*SPARE - Spare *)
                            _769 : REAL; (*SPARE - Spare *)
                            _770 : REAL; (*SPARE - Spare *)
                            _771 : REAL; (*SPARE - Spare *)
                            _772 : REAL; (*SPARE - Spare *)
                            _773 : REAL; (*SPARE - Spare *)
                            _774 : REAL; (*SPARE - Spare *)
                            _775 : REAL; (*SPARE - Spare *)
                            _776 : REAL; (*SPARE - Spare *)
                            _777 : REAL; (*SPARE - Spare *)
                            _778 : REAL; (*SPARE - Spare *)
                            _779 : REAL; (*SPARE - Spare *)
                            _780 : REAL; (*SPARE - Spare *)
                            _781 : REAL; (*SPARE - Spare *)
                            _782 : REAL; (*SPARE - Spare *)
                            _783 : REAL; (*SPARE - Spare *)
                            _784 : REAL; (*SPARE - Spare *)
                            _785 : REAL; (*SPARE - Spare *)
                            _786 : REAL; (*SPARE - Spare *)
                            _787 : REAL; (*SPARE - Spare *)
                            _788 : REAL; (*SPARE - Spare *)
                            _789 : REAL; (*SPARE - Spare *)
                            _790 : REAL; (*SPARE - Spare *)
                            _791 : REAL; (*SPARE - Spare *)
                            _792 : REAL; (*SPARE - Spare *)
                            _793 : REAL; (*SPARE - Spare *)
                            _794 : REAL; (*SPARE - Spare *)
                            _795 : REAL; (*SPARE - Spare *)
                            _796 : REAL; (*SPARE - Spare *)
                            _797 : REAL; (*SPARE - Spare *)
                            _798 : REAL; (*SPARE - Spare *)
                            _799 : REAL; (*SPARE - Spare *)
                            _800 : REAL; (*SPARE - Spare *)
                            _801 : REAL; (*SPARE - Spare *)
                            _802 : REAL; (*SPARE - Spare *)
                            _803 : REAL; (*SPARE - Spare *)
                            _804 : REAL; (*SPARE - Spare *)
                            _805 : REAL; (*SPARE - Spare *)
                            _806 : REAL; (*SPARE - Spare *)
                            _807 : REAL; (*SPARE - Spare *)
                            _808 : REAL; (*SPARE - Spare *)
                            _809 : REAL; (*SPARE - Spare *)
                            _810 : REAL; (*SPARE - Spare *)
                            _811 : REAL; (*SPARE - Spare *)
                            _812 : REAL; (*SPARE - Spare *)
                            _813 : REAL; (*SPARE - Spare *)
                            _814 : REAL; (*SPARE - Spare *)
                            _815 : REAL; (*SPARE - Spare *)
                            _816 : REAL; (*SPARE - Spare *)
                            _817 : REAL; (*SPARE - Spare *)
                            _818 : REAL; (*SPARE - Spare *)
                            _819 : REAL; (*SPARE - Spare *)
                            _820 : REAL; (*SPARE - Spare *)
                            _821 : REAL; (*SPARE - Spare *)
                            _822 : REAL; (*SPARE - Spare *)
                            _823 : REAL; (*SPARE - Spare *)
                            _824 : REAL; (*SPARE - Spare *)
                            _825 : REAL; (*SPARE - Spare *)
                            _826 : REAL; (*SPARE - Spare *)
                            _827 : REAL; (*SPARE - Spare *)
                            _828 : REAL; (*SPARE - Spare *)
                            _829 : REAL; (*SPARE - Spare *)
                            _830 : REAL; (*SPARE - Spare *)
                            _831 : REAL; (*SPARE - Spare *)
                            _832 : REAL; (*SPARE - Spare *)
                            _833 : REAL; (*SPARE - Spare *)
                            _834 : REAL; (*SPARE - Spare *)
                            _835 : REAL; (*SPARE - Spare *)
                            _836 : REAL; (*SPARE - Spare *)
                            _837 : REAL; (*SPARE - Spare *)
                            _838 : REAL; (*SPARE - Spare *)
                            _839 : REAL; (*SPARE - Spare *)
                            _840 : REAL; (*SPARE - Spare *)
                            _841 : REAL; (*SPARE - Spare *)
                            _842 : REAL; (*SPARE - Spare *)
                            _843 : REAL; (*SPARE - Spare *)
                            _844 : REAL; (*SPARE - Spare *)
                            _845 : REAL; (*SPARE - Spare *)
                            _846 : REAL; (*SPARE - Spare *)
                            _847 : REAL; (*SPARE - Spare *)
                            _848 : REAL; (*SPARE - Spare *)
                            _849 : REAL; (*SPARE - Spare *)
                            _850 : REAL; (*SPARE - Spare *)
                            _851 : REAL; (*SPARE - Spare *)
                            _852 : REAL; (*SPARE - Spare *)
                            _853 : REAL; (*SPARE - Spare *)
                            _854 : REAL; (*SPARE - Spare *)
                            _855 : REAL; (*SPARE - Spare *)
                            _856 : REAL; (*SPARE - Spare *)
                            _857 : REAL; (*SPARE - Spare *)
                            _858 : REAL; (*SPARE - Spare *)
                            _859 : REAL; (*SPARE - Spare *)
                            _860 : REAL; (*SPARE - Spare *)
                            _861 : REAL; (*SPARE - Spare *)
                            _862 : REAL; (*SPARE - Spare *)
                            _863 : REAL; (*SPARE - Spare *)
                            _864 : REAL; (*SPARE - Spare *)
                            _865 : REAL; (*SPARE - Spare *)
                            _866 : REAL; (*SPARE - Spare *)
                            _867 : REAL; (*SPARE - Spare *)
                            _868 : REAL; (*SPARE - Spare *)
                            _869 : REAL; (*SPARE - Spare *)
                            _870 : REAL; (*SPARE - Spare *)
                            _871 : REAL; (*SPARE - Spare *)
                            _872 : REAL; (*SPARE - Spare *)
                            _873 : REAL; (*SPARE - Spare *)
                            _874 : REAL; (*SPARE - Spare *)
                            _875 : REAL; (*SPARE - Spare *)
                            _876 : REAL; (*SPARE - Spare *)
                            _877 : REAL; (*SPARE - Spare *)
                            _878 : REAL; (*SPARE - Spare *)
                            _879 : REAL; (*SPARE - Spare *)
                            _880 : REAL; (*SPARE - Spare *)
                            _881 : REAL; (*SPARE - Spare *)
                            _882 : REAL; (*SPARE - Spare *)
                            _883 : REAL; (*SPARE - Spare *)
                            _884 : REAL; (*SPARE - Spare *)
                            _885 : REAL; (*SPARE - Spare *)
                            _886 : REAL; (*SPARE - Spare *)
                            _887 : REAL; (*SPARE - Spare *)
                            _888 : REAL; (*SPARE - Spare *)
                            _889 : REAL; (*SPARE - Spare *)
                            _890 : REAL; (*SPARE - Spare *)
                            _891 : REAL; (*SPARE - Spare *)
                            _892 : REAL; (*SPARE - Spare *)
                            _893 : REAL; (*SPARE - Spare *)
                            _894 : REAL; (*SPARE - Spare *)
                            _895 : REAL; (*SPARE - Spare *)
                            _896 : REAL; (*SPARE - Spare *)
                            _897 : REAL; (*SPARE - Spare *)
                            _898 : REAL; (*SPARE - Spare *)
                            _899 : REAL; (*SPARE - Spare *)
                            _900 : REAL; (*SPARE - Spare *)
                            _901 : REAL; (*SPARE - Spare *)
                            _902 : REAL; (*SPARE - Spare *)
                            _903 : REAL; (*SPARE - Spare *)
                            _904 : REAL; (*SPARE - Spare *)
                            _905 : REAL; (*SPARE - Spare *)
                            _906 : REAL; (*SPARE - Spare *)
                            _907 : REAL; (*SPARE - Spare *)
                            _908 : REAL; (*SPARE - Spare *)
                            _909 : REAL; (*SPARE - Spare *)
                            _910 : REAL; (*SPARE - Spare *)
                            _911 : REAL; (*SPARE - Spare *)
                            _912 : REAL; (*SPARE - Spare *)
                            _913 : REAL; (*SPARE - Spare *)
                            _914 : REAL; (*SPARE - Spare *)
                            _915 : REAL; (*SPARE - Spare *)
                            _916 : REAL; (*SPARE - Spare *)
                            _917 : REAL; (*SPARE - Spare *)
                            _918 : REAL; (*SPARE - Spare *)
                            _919 : REAL; (*SPARE - Spare *)
                            _920 : REAL; (*SPARE - Spare *)
                            _921 : REAL; (*SPARE - Spare *)
                            _922 : REAL; (*SPARE - Spare *)
                            _923 : REAL; (*SPARE - Spare *)
                            _924 : REAL; (*SPARE - Spare *)
                            _925 : REAL; (*SPARE - Spare *)
                            _926 : REAL; (*SPARE - Spare *)
                            _927 : REAL; (*SPARE - Spare *)
                            _928 : REAL; (*SPARE - Spare *)
                            _929 : REAL; (*SPARE - Spare *)
                            _930 : REAL; (*SPARE - Spare *)
                            _931 : REAL; (*SPARE - Spare *)
                            _932 : REAL; (*SPARE - Spare *)
                            _933 : REAL; (*SPARE - Spare *)
                            _934 : REAL; (*SPARE - Spare *)
                            _935 : REAL; (*SPARE - Spare *)
                            _936 : REAL; (*SPARE - Spare *)
                            _937 : REAL; (*SPARE - Spare *)
                            _938 : REAL; (*SPARE - Spare *)
                            _939 : REAL; (*SPARE - Spare *)
                            _940 : REAL; (*SPARE - Spare *)
                            _941 : REAL; (*SPARE - Spare *)
                            _942 : REAL; (*SPARE - Spare *)
                            _943 : REAL; (*SPARE - Spare *)
                            _944 : REAL; (*SPARE - Spare *)
                            _945 : REAL; (*SPARE - Spare *)
                            _946 : REAL; (*SPARE - Spare *)
                            _947 : REAL; (*SPARE - Spare *)
                            _948 : REAL; (*SPARE - Spare *)
                            _949 : REAL; (*SPARE - Spare *)
                            _950 : REAL; (*SPARE - Spare *)
                            _951 : REAL; (*SPARE - Spare *)
                            _952 : REAL; (*SPARE - Spare *)
                            _953 : REAL; (*SPARE - Spare *)
                            _954 : REAL; (*SPARE - Spare *)
                            _955 : REAL; (*SPARE - Spare *)
                            _956 : REAL; (*SPARE - Spare *)
                            _957 : REAL; (*SPARE - Spare *)
                            _958 : REAL; (*SPARE - Spare *)
                            _959 : REAL; (*SPARE - Spare *)
                            _960 : REAL; (*SPARE - Spare *)
                            _961 : REAL; (*SPARE - Spare *)
                            _962 : REAL; (*SPARE - Spare *)
                            _963 : REAL; (*SPARE - Spare *)
                            _964 : REAL; (*SPARE - Spare *)
                            _965 : REAL; (*SPARE - Spare *)
                            _966 : REAL; (*SPARE - Spare *)
                            _967 : REAL; (*SPARE - Spare *)
                            _968 : REAL; (*SPARE - Spare *)
                            _969 : REAL; (*SPARE - Spare *)
                            _970 : REAL; (*SPARE - Spare *)
                            _971 : REAL; (*SPARE - Spare *)
                            _972 : REAL; (*SPARE - Spare *)
                            _973 : REAL; (*SPARE - Spare *)
                            _974 : REAL; (*SPARE - Spare *)
                            _975 : REAL; (*SPARE - Spare *)
                            _976 : REAL; (*SPARE - Spare *)
                            _977 : REAL; (*SPARE - Spare *)
                            _978 : REAL; (*SPARE - Spare *)
                            _979 : REAL; (*SPARE - Spare *)
                            _980 : REAL; (*SPARE - Spare *)
                            _981 : REAL; (*SPARE - Spare *)
                            _982 : REAL; (*SPARE - Spare *)
                            _983 : REAL; (*SPARE - Spare *)
                            _984 : REAL; (*SPARE - Spare *)
                            _985 : REAL; (*SPARE - Spare *)
                            _986 : REAL; (*SPARE - Spare *)
                            _987 : REAL; (*SPARE - Spare *)
                            _988 : REAL; (*SPARE - Spare *)
                            _989 : REAL; (*SPARE - Spare *)
                            _990 : REAL; (*SPARE - Spare *)
                            _991 : REAL; (*SPARE - Spare *)
                            _992 : REAL; (*SPARE - Spare *)
                            _993 : REAL; (*SPARE - Spare *)
                            _994 : REAL; (*SPARE - Spare *)
                            _995 : REAL; (*SPARE - Spare *)
                            _996 : REAL; (*SPARE - Spare *)
                            _997 : REAL; (*SPARE - Spare *)
                            _998 : REAL; (*SPARE - Spare *)
                            _999 : REAL; (*SPARE - Spare *)
        END_STRUCT;
END_TYPE
```
